// TIA Portal V18 export
TYPE "UDT_Store_Holidays"
// stored: IsFailsafeCompliant false
   STRUCT
      UDT_Store_Holidays : Array[0..7] of Date;
   END_STRUCT;
END_TYPE
